TYPE ST_UpdateVehicleReservationDataData :
STRUCT
	sObjectID					: STRING := 'MAIN.fbMMServer';
	sMethodID					: STRING := 'MAIN.fbMMServer#M_UpdateVehicleReservationData';
	iStatus						: INT;
	iNoOfInputArgs				: BYTE := 6;
	iNoOfOutputArgs				: BYTE := 2;
	stInput						: ST_UpdateVehicleReservationDataDataIn;
	stOutput					: ST_UpdateVehicleReservationDataDataOut;
END_STRUCT
END_TYPE

(* stored: Version 1.1.0.1, ProductVersion 3.1.4024.5
   DUT ST_UpdateVehicleReservationDataData: Id {f054530d-0288-45a1-b798-4ebf95d03599} *)
